PROGRAM MAIN
VAR
	
	machineCycle        : machineStation;
	incCommCycle		: incCommStation;
	stackerLoadCycle    : stackerLoadStation;
	stackerUnloadCycle  : stackerUnloadStation;
	insertLoadCycle     : insertLoadStation;
	insertUnloadCycle   : insertUnloadStation;
	roboArmCycle        : roboArmStation;

END_VAR




	machineCycle	   (stBase := Stations.machineStBase,      activeEMG := FALSE,                ioImage := Stations.machineImageIO,
				  		depClear:= DEBUG.machinedClearDep,     syncClear := DEBUG.machinedClearSync);
				
	incCommCycle	   (stBase := Stations.incCommStBase,      activeEMG := Global.emgStopSignal, ioImage := Stations.incCommImageIO,
				        depClear:= DEBUG.incCommClearDep,      syncClear := DEBUG.incCommClearSync);
				 
	stackerLoadCycle   (stBase := Stations.sLoadStBase,        activeEMG := Global.emgStopSignal, ioImage := Stations.sLoadImageIO,
				        depClear:= DEBUG.sLoadClearDep,        syncClear := DEBUG.sLoadClearSync);
				  
	stackerUnloadCycle (stBase := Stations.sUnloadStBase,      activeEMG := Global.emgStopSignal, ioImage := Stations.sUnloadImageIO,
				        depClear:= DEBUG.sUnloadClearDep,      syncClear := DEBUG.sUnloadClearSync);
					
	insertLoadCycle    (stBase := Stations.insertLoadStBase,   activeEMG := Global.emgStopSignal, ioImage := Stations.insertLoadImageIO,
				        depClear:= DEBUG.insertLoadClearDep,   syncClear := DEBUG.insertLoadClearSync);
					
	insertUnloadCycle  (stBase := Stations.insertUnloadStBase, activeEMG := Global.emgStopSignal, ioImage := Stations.insertUnLoadImageIO,
				        depClear:= DEBUG.insertUnloadClearDep, syncClear := DEBUG.insertUnloadClearSync);
					
	roboArmCycle       (stBase := Stations.roboStBase,         activeEMG := Global.emgStopSignal, ioImage := Stations.roboImageIO,
				       depClear:= DEBUG.roboClearDep,          syncClear := DEBUG.roboClearSync);

END_PROGRAM

(* stored: Version 1.1.0.1, ProductVersion 3.1.4024.3
   POU MAIN: Id {94112693-1b8c-4bf4-89c4-cc50028acf18}, SpecialFunc None *)
